// TIA Portal project "Project3" (V15.1)

(* hardware
DEVICE "S7-1200 station_1"  S7-1200 Station
   slot 0: "Rack_0"  S7-1200 Rack  Rack  V1.0
   slot 1: "PLC_1"  CPU 1214C DC/DC/Rly  6ES7 214-1HG40-0XB0  V4.2
*)

// ===== PLC "PLC_1"  CPU 1214C DC/DC/Rly =====

VAR_GLOBAL   // PLC tag table "Default tag table"
   "Tag_1" AT %I0.0 : Bool;
   "Tag_2" AT %Q0.0 : Bool;
   "Tag_3" AT %Q0.1 : Bool;
   "Tag_4" AT %M0.0 : Bool;
   "Tag_5" AT %M0.2 : Bool;
   "Tag_6" AT %M1.0 : Bool;
   "Tag_7" AT %M2.1 : Bool;
   "Tag_8" AT %M3.0 : Bool;
   "Tag_9" AT %M3.1 : Bool;
   "Tag_10" AT %M3.2 : Bool;
   "Tag_11" AT %M3.3 : Bool;
   "Tag_12" AT %M3.4 : Bool;
   "Tag_13" AT %M3.5 : Bool;
   "Tag_14" AT %M3.6 : Bool;
   "Tag_15" AT %M3.7 : Bool;
   "Tag_16" AT %Q1.0 : Bool;
   "rrr" AT %MW10 : Word;
   "Tag_17" AT %QD10 : Time;
   "Tag_18" AT %MD10 : Time;
   "Tag_19" AT %Q0.5 : Bool;
   "Tag_20" AT %Q1.1 : Bool;
   "Tag_21" AT %Q1.2 : Bool;
END_VAR

DATA_BLOCK "D_1"   // DB2
{ S7_Optimized_Access := 'TRUE' }
VERSION : 0.1
   VAR
      "I0.0" : Bool;
      "Q0.0" : Bool;
      "Q0.1" : Bool;
      MD10 : DWord;
   END_VAR
BEGIN
END_DATA_BLOCK

DATA_BLOCK "D_2"   // DB3
{ S7_Optimized_Access := 'TRUE' }
VERSION : 0.1
   VAR
      "Q0.0" : Word := 16#20;
   END_VAR
BEGIN
END_DATA_BLOCK

DATA_BLOCK "Data_block_1"   // DB4
{ S7_Optimized_Access := 'TRUE' }
VERSION : 0.1
   VAR
      "Q0.0" : Bool := True;
      "Q0.1" : Bool;
   END_VAR
BEGIN
END_DATA_BLOCK

DATA_BLOCK "Data_block_2"   // DB5
{ S7_Optimized_Access := 'TRUE' }
VERSION : 0.1
   VAR RETAIN
      "I0.0" : Bool;
      "I0.1" : Bool;
      "I0.2" : Bool;
      "I0.3" : Bool;
      "I0.4" : Bool;
      "I0.1_1" : Bool;
      "I0.2_1" : Bool;
      "I0.3_1" : Bool;
   END_VAR
BEGIN
END_DATA_BLOCK

// folder: System blocks/Program resources

DATA_BLOCK "IEC_Timer_0_DB"   // DB1
{ S7_Optimized_Access := 'TRUE' }
AUTHOR : Simatic
FAMILY : IEC
NAME : IEC_TMR
VERSION : 1.0
// stored: InstanceOfName IEC_TIMER
"IEC_TIMER"
BEGIN
END_DATA_BLOCK

// folder: (top level)

ORGANIZATION_BLOCK "Main"   // OB123, LAD, ProgramCycle
TITLE = "Main Program Sweep (Cycle)"
{ S7_Optimized_Access := 'TRUE' }
VERSION : 0.1
   VAR_INPUT
      Initial_Call : Bool;   // Initial call of this OB
      Remanence : Bool;   // =True, if remanent data are available
   END_VAR
BEGIN

REGION Network 1
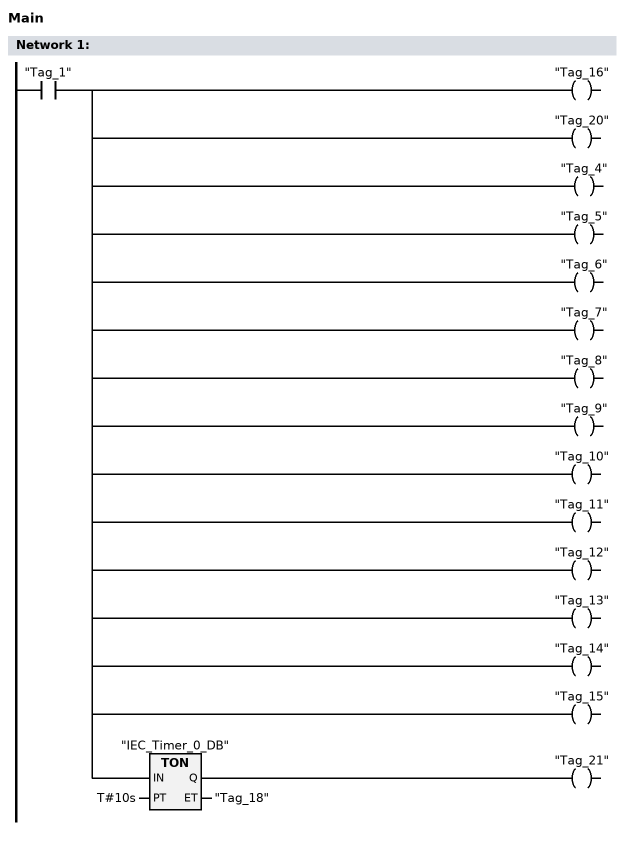
   "Tag_16" := "Tag_1";
   "Tag_20" := "Tag_1";
   "Tag_4" := "Tag_1";
   "Tag_5" := "Tag_1";
   "Tag_6" := "Tag_1";
   "Tag_7" := "Tag_1";
   "Tag_8" := "Tag_1";
   "Tag_9" := "Tag_1";
   "Tag_10" := "Tag_1";
   "Tag_11" := "Tag_1";
   "Tag_12" := "Tag_1";
   "Tag_13" := "Tag_1";
   "Tag_14" := "Tag_1";
   "Tag_15" := "Tag_1";
   "IEC_Timer_0_DB".TON(IN := "Tag_1", PT := T#10s, ET => "Tag_18");
   "Tag_21" := "IEC_Timer_0_DB".Q;
END_REGION
END_ORGANIZATION_BLOCK